FUNCTION HLI3_SetProbingSignal : BOOL
VAR_INPUT
	nHliAxisIdx: INT;
	bProbingSignal: BOOL;
END_VAR


IF NOT HLI3_CheckAxisValid(nHliAxisIdx := nHliAxisIdx) THEN	
	HLI3_SetProbingSignal := FALSE;
	RETURN;
END_IF


gpAx[nHliAxisIdx]^.lr_mc_control.probing_signal.enable_w  := TRUE;
gpAx[nHliAxisIdx]^.lr_mc_control.probing_signal.command_w := bProbingSignal;
HLI3_SetProbingSignal := TRUE;

END_FUNCTION

(* stored: Version 1.1.0.1, ProductVersion 3.1.0.12
   POU HLI3_SetProbingSignal: Id {4969e280-1a3d-43a6-b4bb-220734708a3a} *)
